{attribute 'linkalways'} 
{attribute 'no_explicit_call' := 'This FB is a CLASS and must be accessed using methods or properties'}
{attribute 'enable_dynamic_creation'}
FUNCTION_BLOCK DatatypeAddedEvent EXTENDS Disposable IMPLEMENTS I_DatatypeAddedEvent
VAR
	_target : I_Datatype;
END_VAR

METHOD FB_init : BOOL
VAR_INPUT
	bInitRetains : BOOL; // if TRUE, the retain variables are initialized (warm start / cold start)
	bInCopyCode : BOOL;  // if TRUE, the instance afterwards gets moved into the copy code (online change)
	Target : I_Datatype;
END_VAR
This^._target := Target;
END_METHOD

PROPERTY PUBLIC Target : I_Datatype
GET
Target := _target;
END_GET
END_PROPERTY

END_FUNCTION_BLOCK

(* stored: Version 1.1.0.1, ProductVersion 3.1.4024.12
   POU DatatypeAddedEvent: Id {e097e3af-1371-0557-08f2-bf130a2212b0}, SpecialFunc None
   Folder Constructor: Id {fa19fdc3-58f0-0a1e-3d1a-d5f6c92e1e10}
   Method FB_init: Id {146e1403-47f3-0586-3108-0a79cd6f726a}
   Property Target: Id {ef60201a-0223-07f7-0dcb-61838f798380}
   Get Get: Id {7fe3326d-1006-02ea-30c6-1a08d7643853} *)
